      rq_wait_ft_sensor_steady(2000)
      zero_ftsensor()
      sleep(0.1)
      # end: URCap Program Node
      # begin: URCap Program Node
      #   Source: Robotiq_Copilot, 1.22.1.14215, Robotiq Inc.
      #   Type: Finishing Tool Control
      $ 59 "Start tool"
      set_standard_digital_out(3, True)
      # end: URCap Program Node
      $ 60 "If dried2≟ False "
      if (dried2 ==   False  ):
        $ 61 "Force"
        sleep(0.02)
        zero_ftsensor()
        force_mode(p[0.0,0.0,0.0,0.0,0.0,0.0], [0, 0, 1, 0, 0, 0], [0.0, 0.0, 6.0, 0.0, 0.0, 0.0], 2, [0.1, 0.1, 0.15, 0.3490658503988659, 0.3490658503988659, 0.3490658503988659])
        $ 62 "Conveyor_Move_mm(width-12)" "noBreak"
        Conveyor_Move_mm(width-12)
        $ 63 "Wait SERVER_STATE==1" "noBreak"
        while (not(modbus_get_signal_status("SERVER_STATE")==1)):
          sync()
        end
        $ 64 "moveHeight" "noBreak"
        $ 65 "currentPosition≔get_actual_tcp_pose()" "noBreak"
        global currentPosition=get_actual_tcp_pose()
        $ 66 "newPosition≔pose_add(currentPosition, p[-height/1000,0,0,0,0,0])" "noBreak"
        global newPosition=pose_add(currentPosition, p[-height/1000,0,0,0,0,0])
        $ 67 "newPosition" "noBreak"
        movel(newPosition, a=0.5, v=0.05)
        $ 68 "Conveyor_Move_mm(-width+12)" "noBreak"
        Conveyor_Move_mm(-width+12)
        $ 69 "Wait SERVER_STATE==1" "noBreak"
        while (not(modbus_get_signal_status("SERVER_STATE")==1)):
          sync()
        end
        $ 70 "moveHeight" "noBreak"
        $ 71 "currentPosition≔get_actual_tcp_pose()" "noBreak"
        global currentPosition=get_actual_tcp_pose()
        $ 72 "newPosition≔pose_add(currentPosition, p[height/1000,0,0,0,0,0])" "noBreak"
        global newPosition=pose_add(currentPosition, p[height/1000,0,0,0,0,0])
        $ 73 "newPosition" "noBreak"
        movel(newPosition, a=0.5, v=0.05)
        # begin: URCap Program Node
        #   Source: Robotiq_Copilot, 1.22.1.14215, Robotiq Inc.
        #   Type: Finishing Tool Control
        $ 74 "Stop tool" "noBreak"
        set_standard_digital_out(3, False)
        # end: URCap Program Node
        end_force_mode()
        stopl(5.0)
      else:
        $ 75 "Else" "noBreak"
        $ 76 "Force"
        sleep(0.02)
        zero_ftsensor()
        force_mode(p[0.0,0.0,0.0,0.0,0.0,0.0], [0, 0, 1, 0, 0, 0], [0.0, 0.0, 6.0, 0.0, 0.0, 0.0], 2, [0.1, 0.1, 0.15, 0.3490658503988659, 0.3490658503988659, 0.3490658503988659])
        $ 77 "Conveyor_Move_mm(width-12)" "noBreak"
        Conveyor_Move_mm(width-12)
        $ 78 "Wait SERVER_STATE==1" "noBreak"
        while (not(modbus_get_signal_status("SERVER_STATE")==1)):
          sync()
        end
        $ 79 "moveHeight" "noBreak"
        $ 80 "currentPosition≔get_actual_tcp_pose()" "noBreak"
        global currentPosition=get_actual_tcp_pose()
        $ 81 "newPosition≔pose_add(currentPosition, p[-height/1000,0,0,0,0,0])" "noBreak"
        global newPosition=pose_add(currentPosition, p[-height/1000,0,0,0,0,0])
        $ 82 "newPosition" "noBreak"
        movel(newPosition, a=0.5, v=0.05)
        $ 83 "Conveyor_Move_mm(-width+12)" "noBreak"
        Conveyor_Move_mm(-width+12)
        $ 84 "Wait SERVER_STATE==1" "noBreak"
        while (not(modbus_get_signal_status("SERVER_STATE")==1)):
          sync()
        end
        $ 85 "moveHeight" "noBreak"
        $ 86 "currentPosition≔get_actual_tcp_pose()" "noBreak"
        global currentPosition=get_actual_tcp_pose()
        $ 87 "newPosition≔pose_add(currentPosition, p[height/1000,0,0,0,0,0])" "noBreak"
        global newPosition=pose_add(currentPosition, p[height/1000,0,0,0,0,0])
        $ 88 "newPosition" "noBreak"
        movel(newPosition, a=0.5, v=0.05)
        # begin: URCap Program Node
        #   Source: Robotiq_Copilot, 1.22.1.14215, Robotiq Inc.
        #   Type: Finishing Tool Control
        $ 89 "Stop tool" "noBreak"
        set_standard_digital_out(3, False)
        # end: URCap Program Node
        end_force_mode()
        stopl(5.0)
      end
      $ 90 "MoveJ"
      $ 91 "Sand_Base" "breakAfter"
      movej(get_inverse_kin(Sand_Base_p, qnear=Sand_Base_q), a=1.3962634015954636, v=1.0471975511965976)
      $ 92 "45 Sand"
      $ 93 "If JOB == 3"
      if (modbus_get_signal_status("JOB") == 3):
        $ 94 "Conveyor_Move_mm((width-12)/3)"
        Conveyor_Move_mm((width-12)/3)
        $ 95 "Wait SERVER_STATE==1"
        while (not(modbus_get_signal_status("SERVER_STATE")==1)):
          sync()
        end
        $ 96 "MoveL"
        $ 97 "Direction: Base Z+"
        global move_thread_flag_97=0
        thread move_thread_97():
          enter_critical
          move_thread_flag_97 = 1
          local towardsPos=calculate_point_to_move_towards(p[0.0,0.0,0.0,0.0,0.0,0.0], [0.0,0.0,1.0], 1000.0)
          movel(towardsPos, a=0.5, v=0.05)
          move_thread_flag_97 = 2
          exit_critical
        end
        move_thread_flag_97 = 0
        move_thread_han_97 = run move_thread_97()
        while (True):
          local targetTcpDirection=get_target_tcp_speed()
          local stepsToRetract=tool_contact(direction=targetTcpDirection)
          if (stepsToRetract > 0):
            kill move_thread_han_97
            stopl(3.0)
            local backTrackMovement=get_actual_joint_positions_history(stepsToRetract)
            local contactPose=get_forward_kin(backTrackMovement)
            local posDir=[targetTcpDirection[0],targetTcpDirection[1],targetTcpDirection[2]]
            local retractTo=contactPose
            if (norm(posDir) > 1e-6):
              local normalizedPosDir=normalize(posDir)
              local additionalRetraction=p[normalizedPosDir[0] * 0.0, normalizedPosDir[1] * 0.0, normalizedPosDir[2] * 0.0, 0, 0, 0]
              retractTo = pose_sub(contactPose, additionalRetraction)
            end
            movel(retractTo, a=3.0, v=0.1)
            $ 98 "Until (tool_contact_detection)"
            break
          end
          sync()
        end
        # begin: URCap Program Node
        #   Source: Robotiq_Copilot, 1.22.1.14215, Robotiq Inc.
        #   Type: Finishing Tool Control
        $ 99 "Start tool"
        set_standard_digital_out(3, True)
        # end: URCap Program Node
        $ 100 "Force"
        sleep(0.02)
        zero_ftsensor()
        force_mode(p[0.0,0.0,0.0,0.0,0.0,0.0], [0, 0, 1, 0, 0, 0], [0.0, 0.0, 7.0, 0.0, 0.0, 0.0], 2, [0.1, 0.1, 0.15, 0.3490658503988659, 0.3490658503988659, 0.3490658503988659])
        $ 101 "moveHeight" "noBreak"
        $ 102 "currentPosition≔get_actual_tcp_pose()" "noBreak"
        global currentPosition=get_actual_tcp_pose()
        $ 103 "newPosition≔pose_add(currentPosition, p[-height/1000,0,0,0,0,0])" "noBreak"
        global newPosition=pose_add(currentPosition, p[-height/1000,0,0,0,0,0])
        $ 104 "newPosition" "noBreak"
        set_tcp(p[0.0010032816279412216,0.1255407840271643,0.10415400799666161,-0.7853981633974483,0.0,0.0])
        movel(newPosition, a=0.5, v=0.05)
        # begin: URCap Program Node
        #   Source: Robotiq_Copilot, 1.22.1.14215, Robotiq Inc.
        #   Type: Finishing Tool Control
        $ 105 "Stop tool" "noBreak"
        set_standard_digital_out(3, False)
        # end: URCap Program Node
        end_force_mode()
        stopl(5.0)
        $ 106 "Direction: Base Z-"
        global move_thread_flag_106=0
        thread move_thread_106():
          enter_critical
          move_thread_flag_106 = 1
          local towardsPos=calculate_point_to_move_towards(p[0.0,0.0,0.0,0.0,0.0,0.0], [0.0,0.0,-1.0], 0.02)
          movel(towardsPos, a=0.5, v=0.05)
          move_thread_flag_106 = 2
          exit_critical
        end
        move_thread_flag_106 = 0
        move_thread_han_106 = run move_thread_106()
        while (True):
          sleep(1.0E-10)
          if (move_thread_flag_106 > 1):
            join move_thread_han_106
            $ 107 "Until (distance)"
            break
          end
          sync()
        end
        $ 108 "Conveyor_Move_mm((width-12)/3)"
        Conveyor_Move_mm((width-12)/3)
        $ 109 "Wait SERVER_STATE==1"
        while (not(modbus_get_signal_status("SERVER_STATE")==1)):
          sync()
        end
        $ 110 "Direction: Base Z+"
        global move_thread_flag_110=0
        thread move_thread_110():
          enter_critical
          move_thread_flag_110 = 1
          local towardsPos=calculate_point_to_move_towards(p[0.0,0.0,0.0,0.0,0.0,0.0], [0.0,0.0,1.0], 1000.0)
          movel(towardsPos, a=0.5, v=0.05)
          move_thread_flag_110 = 2
          exit_critical
        end
        move_thread_flag_110 = 0
        move_thread_han_110 = run move_thread_110()
        while (True):
          local targetTcpDirection=get_target_tcp_speed()
          local stepsToRetract=tool_contact(direction=targetTcpDirection)
          if (stepsToRetract > 0):
            kill move_thread_han_110
            stopl(3.0)
            local backTrackMovement=get_actual_joint_positions_history(stepsToRetract)
            local contactPose=get_forward_kin(backTrackMovement)
            local posDir=[targetTcpDirection[0],targetTcpDirection[1],targetTcpDirection[2]]
            local retractTo=contactPose
            if (norm(posDir) > 1e-6):
              local normalizedPosDir=normalize(posDir)
              local additionalRetraction=p[normalizedPosDir[0] * 0.0, normalizedPosDir[1] * 0.0, normalizedPosDir[2] * 0.0, 0, 0, 0]
              retractTo = pose_sub(contactPose, additionalRetraction)
            end
            movel(retractTo, a=3.0, v=0.1)
            $ 111 "Until (tool_contact_detection)"
            break
          end
          sync()
        end
        $ 112 "Force"
        sleep(0.02)
        zero_ftsensor()
        force_mode(p[0.0,0.0,0.0,0.0,0.0,0.0], [0, 0, 1, 0, 0, 0], [0.0, 0.0, 7.0, 0.0, 0.0, 0.0], 2, [0.1, 0.1, 0.15, 0.3490658503988659, 0.3490658503988659, 0.3490658503988659])
        # begin: URCap Program Node
        #   Source: Robotiq_Copilot, 1.22.1.14215, Robotiq Inc.
        #   Type: Finishing Tool Control
        $ 113 "Start tool" "noBreak"
        set_standard_digital_out(3, True)
        # end: URCap Program Node
        $ 114 "moveHeight" "noBreak"
        $ 115 "currentPosition≔get_actual_tcp_pose()" "noBreak"
        global currentPosition=get_actual_tcp_pose()
        $ 116 "newPosition≔pose_add(currentPosition, p[height/1000,0,0,0,0,0])" "noBreak"
        global newPosition=pose_add(currentPosition, p[height/1000,0,0,0,0,0])
        $ 117 "newPosition" "noBreak"
        set_tcp(p[0.0010032816279412216,0.1255407840271643,0.10415400799666161,-0.7853981633974483,0.0,0.0])
        movel(newPosition, a=0.5, v=0.05)
        # begin: URCap Program Node
        #   Source: Robotiq_Copilot, 1.22.1.14215, Robotiq Inc.
        #   Type: Finishing Tool Control
        $ 118 "Stop tool" "noBreak"
        set_standard_digital_out(3, False)
        # end: URCap Program Node
        end_force_mode()
        stopl(5.0)
        $ 119 "Direction: Base Z-"
        global move_thread_flag_119=0
        thread move_thread_119():
          enter_critical
          move_thread_flag_119 = 1
          local towardsPos=calculate_point_to_move_towards(p[0.0,0.0,0.0,0.0,0.0,0.0], [0.0,0.0,-1.0], 0.02)
          movel(towardsPos, a=0.5, v=0.05)
          move_thread_flag_119 = 2
          exit_critical
        end
        move_thread_flag_119 = 0
        move_thread_han_119 = run move_thread_119()
        while (True):
          sleep(1.0E-10)
          if (move_thread_flag_119 > 1):
            join move_thread_han_119
            $ 120 "Until (distance)"
            break
          end
          sync()
        end
        $ 121 "Conveyor_Move_mm(-(width-12)*2/3)"
        Conveyor_Move_mm(-(width-12)*2/3)
        $ 122 "Wait SERVER_STATE==1"
        while (not(modbus_get_signal_status("SERVER_STATE")==1)):
          sync()
        end
      end
      $ 123 "SC 3 and 4 Sand"
      $ 124 "If JOB == 5 or JOB == 6"
      if (modbus_get_signal_status("JOB") == 5 or modbus_get_signal_status("JOB") == 6):
        $ 125 "Conveyor_Move_mm((width-12)/2)"
        Conveyor_Move_mm((width-12)/2)
        $ 126 "Wait SERVER_STATE==1"
        while (not(modbus_get_signal_status("SERVER_STATE")==1)):
          sync()
        end
        $ 127 "MoveL"
        $ 128 "Direction: Base X-"
        global move_thread_flag_128=0
        thread move_thread_128():
          enter_critical
          move_thread_flag_128 = 1
          local towardsPos=calculate_point_to_move_towards(p[0.0,0.0,0.0,0.0,0.0,0.0], [-1.0,0.0,0.0], 0.085)
          movel(towardsPos, a=0.5, v=0.05)
          move_thread_flag_128 = 2
          exit_critical
        end
        move_thread_flag_128 = 0
        move_thread_han_128 = run move_thread_128()
        while (True):
          sleep(1.0E-10)
          if (move_thread_flag_128 > 1):
            join move_thread_han_128
            $ 129 "Until (distance)"
            break
          end
          sync()
        end
        $ 130 "Direction: Base Z+"
        global move_thread_flag_130=0
        thread move_thread_130():
          enter_critical
          move_thread_flag_130 = 1
          local towardsPos=calculate_point_to_move_towards(p[0.0,0.0,0.0,0.0,0.0,0.0], [0.0,0.0,1.0], 1000.0)
          movel(towardsPos, a=0.5, v=0.05)
          move_thread_flag_130 = 2
          exit_critical
        end
        move_thread_flag_130 = 0
        move_thread_han_130 = run move_thread_130()
        while (True):
          local targetTcpDirection=get_target_tcp_speed()
          local stepsToRetract=tool_contact(direction=targetTcpDirection)
          if (stepsToRetract > 0):
            kill move_thread_han_130
            stopl(3.0)
            local backTrackMovement=get_actual_joint_positions_history(stepsToRetract)
            local contactPose=get_forward_kin(backTrackMovement)
            local posDir=[targetTcpDirection[0],targetTcpDirection[1],targetTcpDirection[2]]
            local retractTo=contactPose
            if (norm(posDir) > 1e-6):
              local normalizedPosDir=normalize(posDir)
              local additionalRetraction=p[normalizedPosDir[0] * 0.0, normalizedPosDir[1] * 0.0, normalizedPosDir[2] * 0.0, 0, 0, 0]
              retractTo = pose_sub(contactPose, additionalRetraction)
            end
            movel(retractTo, a=3.0, v=0.1)
            $ 131 "Until (tool_contact_detection)"
            break
          end
          sync()
        end
        # begin: URCap Program Node
        #   Source: Robotiq_Copilot, 1.22.1.14215, Robotiq Inc.
        #   Type: Finishing Tool Control
        $ 132 "Start tool"
        set_standard_digital_out(3, True)
        # end: URCap Program Node
        $ 133 "Force"
        sleep(0.02)
        zero_ftsensor()
        force_mode(p[0.0,0.0,0.0,0.0,0.0,0.0], [0, 0, 1, 0, 0, 0], [0.0, 0.0, 10.0, 0.0, 0.0, 0.0], 2, [0.1, 0.1, 0.15, 0.3490658503988659, 0.3490658503988659, 0.3490658503988659])
        $ 134 "Direction: Base X-" "noBreak"
        global move_thread_flag_134=0
        thread move_thread_134():
          enter_critical
          move_thread_flag_134 = 1
          local towardsPos=calculate_point_to_move_towards(p[0.0,0.0,0.0,0.0,0.0,0.0], [-1.0,0.0,0.0], 0.08)
          movel(towardsPos, a=0.5, v=0.05)
          move_thread_flag_134 = 2
          exit_critical
        end
        move_thread_flag_134 = 0
        move_thread_han_134 = run move_thread_134()
        while (True):
          sleep(1.0E-10)
          if (move_thread_flag_134 > 1):
            join move_thread_han_134
            $ 135 "Until (distance)" "noBreak"
            break
          end
          sync()
        end
        # begin: URCap Program Node
        #   Source: Robotiq_Copilot, 1.22.1.14215, Robotiq Inc.
        #   Type: Finishing Tool Control
        $ 136 "Stop tool" "noBreak"
        set_standard_digital_out(3, False)
        # end: URCap Program Node
        end_force_mode()
        stopl(5.0)
        $ 137 "Direction: Base Z-"
        global move_thread_flag_137=0
        thread move_thread_137():
          enter_critical
          move_thread_flag_137 = 1
          local towardsPos=calculate_point_to_move_towards(p[0.0,0.0,0.0,0.0,0.0,0.0], [0.0,0.0,-1.0], 0.05)
          movel(towardsPos, a=0.5, v=0.05)
          move_thread_flag_137 = 2
          exit_critical
        end
        move_thread_flag_137 = 0
        move_thread_han_137 = run move_thread_137()
        while (True):
          sleep(1.0E-10)
          if (move_thread_flag_137 > 1):
            join move_thread_han_137
            $ 138 "Until (distance)"
            break
          end
          sync()
        end
        $ 139 "Conveyor_Move_mm(-(width-12)/2)"
        Conveyor_Move_mm(-(width-12)/2)
        $ 140 "Wait SERVER_STATE==1"
        while (not(modbus_get_signal_status("SERVER_STATE")==1)):
          sync()
        end
      end
      $ 141 "Spray Vertical"
      $ 142 "MoveJ"
      $ 143 "Spray_Base" "breakAfter"
      set_tcp(p[0.06314273891748035,-0.10788249600106846,0.08439511317031662,0.6139431255689367,0.6139431255689367,-1.4821898202742554])
      movej(get_inverse_kin(Spray_Base_p, qnear=Spray_Base_q), a=1.3962634015954636, v=1.0471975511965976)
      $ 144 "If JOB == 2"
      if (modbus_get_signal_status("JOB") == 2):
        $ 145 "MoveL"
        $ 146 "Direction: Base Z+"
        global move_thread_flag_146=0
        thread move_thread_146():
          enter_critical
          move_thread_flag_146 = 1
          local towardsPos=calculate_point_to_move_towards(p[0.0,0.0,0.0,0.0,0.0,0.0], [0.0,0.0,1.0], 0.1)
          movel(towardsPos, a=1.2, v=0.25)
          move_thread_flag_146 = 2
          exit_critical
        end
        move_thread_flag_146 = 0
        move_thread_han_146 = run move_thread_146()
        while (True):
          sleep(1.0E-10)
          if (move_thread_flag_146 > 1):
            join move_thread_han_146
            $ 147 "Until (distance)"
            break
          end
          sync()
        end
      end
      $ 148 "If JOB == 7"
      if (modbus_get_signal_status("JOB") == 7):
        $ 149 "MoveL"
        $ 150 "Direction: Base Z+"
        global move_thread_flag_150=0
        thread move_thread_150():
          enter_critical
          move_thread_flag_150 = 1
          local towardsPos=calculate_point_to_move_towards(p[0.0,0.0,0.0,0.0,0.0,0.0], [0.0,0.0,1.0], 0.2)
          movel(towardsPos, a=1.2, v=0.25)
          move_thread_flag_150 = 2
          exit_critical
        end
        move_thread_flag_150 = 0
        move_thread_han_150 = run move_thread_150()
        while (True):
          sleep(1.0E-10)
          if (move_thread_flag_150 > 1):
            join move_thread_han_150
            $ 151 "Until (distance)"
            break
          end
          sync()
        end
      end
      $ 152 "Set SprayerOn=On"
      set_standard_digital_out(5, True)
      $ 153 "MoveL"
      $ 154 "Conveyor_Move_mm(width-12)"
      Conveyor_Move_mm(width-12)
      $ 155 "Wait SERVER_STATE==1"
      while (not(modbus_get_signal_status("SERVER_STATE")==1)):
        sync()
      end
      $ 156 "moveHeight"
      $ 157 "currentPosition≔get_actual_tcp_pose()"
      global currentPosition=get_actual_tcp_pose()
      $ 158 "newPosition≔pose_add(currentPosition, p[-height/1000,0,0,0,0,0])"
      global newPosition=pose_add(currentPosition, p[-height/1000,0,0,0,0,0])
      $ 159 "newPosition" "breakAfter"
      movel(newPosition, a=0.5, v=0.05)
      $ 160 "Conveyor_Move_mm(-width+12)"
      Conveyor_Move_mm(-width+12)
      $ 161 "Wait SERVER_STATE==1"
      while (not(modbus_get_signal_status("SERVER_STATE")==1)):
        sync()
      end
      $ 162 "moveHeight"
      $ 163 "currentPosition≔get_actual_tcp_pose()"
      global currentPosition=get_actual_tcp_pose()
      $ 164 "newPosition≔pose_add(currentPosition, p[height/1000,0,0,0,0,0])"
      global newPosition=pose_add(currentPosition, p[height/1000,0,0,0,0,0])
      $ 165 "newPosition" "breakAfter"
      movel(newPosition, a=0.5, v=0.05)
      $ 166 "Set SprayerOn=Off"
      set_standard_digital_out(5, False)
      $ 167 "MoveJ"
      $ 168 "Spray_Base" "breakAfter"
      movej(get_inverse_kin(Spray_Base_p, qnear=Spray_Base_q), a=1.3962634015954636, v=1.0471975511965976)
      $ 169 "45 Spray"
      $ 170 "If JOB == 3"
      if (modbus_get_signal_status("JOB") == 3):
        $ 171 "MoveJ"
        $ 172 "Spray_Base" "breakAfter"
        set_tcp(p[0.06314273891748035,-0.10788249600106846,0.08439511317031662,0.6139431255689367,0.6139431255689367,-1.4821898202742554])
        movej(get_inverse_kin(Spray_Base_p, qnear=Spray_Base_q), a=1.3962634015954636, v=1.0471975511965976)
        $ 173 "MoveL"
        $ 174 "Conveyor_Move_mm(width/3)"
        Conveyor_Move_mm(width/3)
        $ 175 "Wait SERVER_STATE==1"
        while (not(modbus_get_signal_status("SERVER_STATE")==1)):
          sync()
        end
        $ 176 "Set SprayerOn=On"
        set_standard_digital_out(5, True)
        $ 177 "moveHeight"
        $ 178 "currentPosition≔get_actual_tcp_pose()"
        global currentPosition=get_actual_tcp_pose()
        $ 179 "newPosition≔pose_add(currentPosition, p[-height/1000,0,0,0,0,0])"
        global newPosition=pose_add(currentPosition, p[-height/1000,0,0,0,0,0])
        $ 180 "newPosition" "breakAfter"
        movel(newPosition, a=0.5, v=0.05)
        $ 181 "Set SprayerOn=Off"
        set_standard_digital_out(5, False)
        $ 182 "Conveyor_Move_mm(width/3)"
        Conveyor_Move_mm(width/3)
        $ 183 "Wait SERVER_STATE==1"
        while (not(modbus_get_signal_status("SERVER_STATE")==1)):
          sync()
        end
        $ 184 "Set SprayerOn=On"
        set_standard_digital_out(5, True)
        $ 185 "moveHeight"
        $ 186 "currentPosition≔get_actual_tcp_pose()"
        global currentPosition=get_actual_tcp_pose()
        $ 187 "newPosition≔pose_add(currentPosition, p[height/1000,0,0,0,0,0])"
        global newPosition=pose_add(currentPosition, p[height/1000,0,0,0,0,0])
        $ 188 "newPosition" "breakAfter"
        movel(newPosition, a=0.5, v=0.05)
        $ 189 "Set SprayerOn=Off"
        set_standard_digital_out(5, False)
        $ 190 "MoveJ"
        $ 191 "Spray_Base" "breakAfter"
        movej(get_inverse_kin(Spray_Base_p, qnear=Spray_Base_q), a=1.3962634015954636, v=1.0471975511965976)
      end
      $ 192 "SC 3 and 4 Spray"
      $ 193 "If JOB == 5 or JOB == 6"
      if (modbus_get_signal_status("JOB") == 5 or modbus_get_signal_status("JOB") == 6):
        $ 194 "MoveJ"
        $ 195 "Spray_Base" "breakAfter"
        set_tcp(p[0.06314273891748035,-0.10788249600106846,0.08439511317031662,0.6139431255689367,0.6139431255689367,-1.4821898202742554])
        movej(get_inverse_kin(Spray_Base_p, qnear=Spray_Base_q), a=1.3962634015954636, v=1.0471975511965976)
        $ 196 "Conveyor_Move_mm((width-12)/2)"
        Conveyor_Move_mm((width-12)/2)
        $ 197 "Wait SERVER_STATE==1"
        while (not(modbus_get_signal_status("SERVER_STATE")==1)):
          sync()
        end
        $ 198 "MoveL"
        $ 199 "Direction: Base X-"
        global move_thread_flag_199=0
        thread move_thread_199():
          enter_critical
          move_thread_flag_199 = 1
          local towardsPos=calculate_point_to_move_towards(p[0.0,0.0,0.0,0.0,0.0,0.0], [-1.0,0.0,0.0], 0.012)
          movel(towardsPos, a=0.5, v=0.05)
          move_thread_flag_199 = 2
          exit_critical
        end
        move_thread_flag_199 = 0
        move_thread_han_199 = run move_thread_199()
        while (True):
          sleep(1.0E-10)
          if (move_thread_flag_199 > 1):
            join move_thread_han_199
            $ 200 "Until (distance)"
            break
          end
          sync()
        end
        $ 201 "Set SprayerOn=On"
        set_standard_digital_out(5, True)
        $ 202 "Direction: Base X-"
        global move_thread_flag_202=0
        thread move_thread_202():
          enter_critical
          move_thread_flag_202 = 1
          local towardsPos=calculate_point_to_move_towards(p[0.0,0.0,0.0,0.0,0.0,0.0], [-1.0,0.0,0.0], 0.21)
          movel(towardsPos, a=0.5, v=0.05)
          move_thread_flag_202 = 2
          exit_critical
        end
        move_thread_flag_202 = 0
        move_thread_han_202 = run move_thread_202()
        while (True):
          sleep(1.0E-10)
          if (move_thread_flag_202 > 1):
            join move_thread_han_202
            $ 203 "Until (distance)"
            break
          end
          sync()
        end
        $ 204 "Set SprayerOn=Off"
        set_standard_digital_out(5, False)
        $ 205 "Conveyor_Move_mm(-(width-12)/2)"
        Conveyor_Move_mm(-(width-12)/2)
        $ 206 "Wait SERVER_STATE==1"
        while (not(modbus_get_signal_status("SERVER_STATE")==1)):
          sync()
        end
      end
      $ 207 "Cube"
      $ 208 "If JOB==1"
      if (modbus_get_signal_status("JOB")==1):
        $ 209 "Spray Horizontal"
        $ 210 "MoveJ"
        $ 211 "Waypoint_1" "breakAfter"
        set_tcp(p[0.06314273891748035,-0.10788249600106846,0.08439511317031662,0.6139431255689367,0.6139431255689367,-1.4821898202742554])
        movej(get_inverse_kin(Waypoint_1_p, qnear=Waypoint_1_q), a=1.3962634015954636, v=1.0471975511965976)
        $ 212 "Set SprayerOn=On"
        set_standard_digital_out(5, True)
        $ 213 "Conveyor_Move_mm(width-12)"
        Conveyor_Move_mm(width-12)
        $ 214 "Wait SERVER_STATE==1"
        while (not(modbus_get_signal_status("SERVER_STATE")==1)):
          sync()
        end
        $ 215 "Set SprayerOn=Off"
        set_standard_digital_out(5, False)
        $ 216 "Waypoint_2" "breakAfter"
        set_tcp(p[0.06314273891748035,-0.10788249600106846,0.08439511317031662,0.6139431255689367,0.6139431255689367,-1.4821898202742554])
        movej(get_inverse_kin(Waypoint_2_p, qnear=Waypoint_2_q), a=1.3962634015954636, v=1.0471975511965976)
        $ 217 "MoveL"
        $ 218 "Set SprayerOn=On"
        set_standard_digital_out(5, True)
        $ 219 "moveHeight"
        $ 220 "currentPosition≔get_actual_tcp_pose()"
        global currentPosition=get_actual_tcp_pose()
        $ 221 "newPosition≔pose_add(currentPosition, p[-height/1000,0,0,0,0,0])"
        global newPosition=pose_add(currentPosition, p[-height/1000,0,0,0,0,0])
        $ 222 "newPosition" "breakAfter"
        movel(newPosition, a=0.5, v=0.05)
        $ 223 "Set SprayerOn=Off"
        set_standard_digital_out(5, False)
        $ 224 "Conveyor_Move_mm(-width+12)"
        Conveyor_Move_mm(-width+12)
        $ 225 "Waypoint_3" "breakAfter"
        set_tcp(p[0.06314273891748035,-0.10788249600106846,0.08439511317031662,0.6139431255689367,0.6139431255689367,-1.4821898202742554])
        movej(get_inverse_kin(Waypoint_3_p, qnear=Waypoint_3_q), a=1.3962634015954636, v=1.0471975511965976)
        $ 226 "Wait SERVER_STATE==1"
        while (not(modbus_get_signal_status("SERVER_STATE")==1)):
          sync()
        end
        $ 227 "MoveL"
        $ 228 "Set SprayerOn=On"
        set_standard_digital_out(5, True)
        $ 229 "moveHeight"
        $ 230 "currentPosition≔get_actual_tcp_pose()"
        global currentPosition=get_actual_tcp_pose()
        $ 231 "newPosition≔pose_add(currentPosition, p[height/1000,0,0,0,0,0])"
        global newPosition=pose_add(currentPosition, p[height/1000,0,0,0,0,0])
        $ 232 "newPosition" "breakAfter"
        movel(newPosition, a=0.5, v=0.05)
        $ 233 "Set SprayerOn=Off"
        set_standard_digital_out(5, False)
      end
      $ 234 "MoveJ"
      $ 235 "Sand_Base" "breakAfter"
      set_tcp(p[0.0010032816279412216,0.1255407840271643,0.10415400799666161,-0.7853981633974483,0.0,0.0])
      movej(get_inverse_kin(Sand_Base_p, qnear=Sand_Base_q), a=1.3962634015954636, v=1.0471975511965976)
      $ 236 "Clean Spray"
      $ 237 "MoveJ"
      $ 238 "Sand_Base" "breakAfter"
      set_tcp(p[0.0010032816279412216,0.1255407840271643,0.10415400799666161,-0.7853981633974483,0.0,0.0])
      movej(get_inverse_kin(Sand_Base_p, qnear=Sand_Base_q), a=1.3962634015954636, v=1.0471975511965976)
      $ 239 "Clean_Brush" "breakAfter"
      set_tcp(p[0.0010032816279412216,0.1255407840271643,0.10415400799666161,-0.7853981633974483,0.0,0.0])
      movej(get_inverse_kin(Clean_Brush_p, qnear=Clean_Brush_q), a=1.3962634015954636, v=1.0471975511965976)
      $ 240 "MoveL"
      $ 241 "Direction: Base Z+"
      global move_thread_flag_241=0
      thread move_thread_241():
        enter_critical
        move_thread_flag_241 = 1
        local towardsPos=calculate_point_to_move_towards(p[0.0,0.0,0.0,0.0,0.0,0.0], [0.0,0.0,1.0], 1000.0)
        movel(towardsPos, a=0.5, v=0.05)
        move_thread_flag_241 = 2
        exit_critical
      end
      move_thread_flag_241 = 0
      move_thread_han_241 = run move_thread_241()
      while (True):
        local targetTcpDirection=get_target_tcp_speed()
        local stepsToRetract=tool_contact(direction=targetTcpDirection)
        if (stepsToRetract > 0):
          kill move_thread_han_241
          stopl(0.5)
          local backTrackMovement=get_actual_joint_positions_history(stepsToRetract)
          local contactPose=get_forward_kin(backTrackMovement)
          local posDir=[targetTcpDirection[0],targetTcpDirection[1],targetTcpDirection[2]]
          local retractTo=contactPose
          if (norm(posDir) > 1e-6):
            local normalizedPosDir=normalize(posDir)
            local additionalRetraction=p[normalizedPosDir[0] * 0.003, normalizedPosDir[1] * 0.003, normalizedPosDir[2] * 0.003, 0, 0, 0]
            retractTo = pose_sub(contactPose, additionalRetraction)
          end
          movel(retractTo, a=0.5, v=0.1)
          $ 242 "Until (tool_contact_detection)"
          break
        end
        sync()
      end
      $ 243 "Wait: 1.0"
      sleep(1.0)
      $ 244 "Set BRUSH_ON_LOCAL= True "
      modbus_set_output_signal("BRUSH_ON_LOCAL",   True  )
      $ 245 "timer_brush: Start"
      timer_brush_is_counting = True
      $ 246 "If dried2≟ False "
      if (dried2 ==   False  ):
        $ 247 "Dry"
        $ 248 "timer_dry: Start"
        timer_dry_is_counting = True
        $ 249 "Conveyor_Move_mm(width+500)"
        Conveyor_Move_mm(width+500)
        $ 250 "Wait SERVER_STATE==1"
        while (not(modbus_get_signal_status("SERVER_STATE")==1)):
          sync()
        end
        $ 251 "Loop timer_dry<165"
        while (timer_dry<165):
          $ 252 "Conveyor_Move_mm(-(width/2))"
          Conveyor_Move_mm(-(width/2))
          $ 253 "Wait SERVER_STATE==1"
          while (not(modbus_get_signal_status("SERVER_STATE")==1)):
            sync()
          end
          $ 254 "Conveyor_Move_mm(width/2)"
          Conveyor_Move_mm(width/2)
          $ 255 "Wait SERVER_STATE==1"
          while (not(modbus_get_signal_status("SERVER_STATE")==1)):
            sync()
          end
        end
        $ 256 "Move_Continuous('reverse')"
        Move_Continuous("reverse")
        $ 257 "Wait WORK_AT_ZERO=HI"
        while (modbus_get_signal_status("WORK_AT_ZERO") == False):
          sync()
        end
        $ 258 "Wait WORK_AT_ZERO=LO"
        while (modbus_get_signal_status("WORK_AT_ZERO") == True):
          sync()
        end
        $ 259 "Move_Continuous('forward')"
        Move_Continuous("forward")
        $ 260 "Wait WORK_AT_ZERO=HI"
        while (modbus_get_signal_status("WORK_AT_ZERO") == False):
          sync()
        end
        $ 261 "dried2≔ True "
        global dried2=  True
        $ 262 "timer_dry: Stop"
        timer_dry_is_counting = False
        $ 263 "timer_dry: Reset"
        timer_dry = 0
        $ 264 "Move_Idle()"
        Move_Idle()
      else:
        $ 265 "Else" "noBreak"
        $ 266 "Unload Workpiece"
        $ 267 "Move_Continuous('forward')"
        Move_Continuous("forward")
        $ 268 "Wait OFFLOAD=HI"
        while (modbus_get_signal_status("OFFLOAD") == False):
          sync()
        end
        $ 269 "Wait OFFLOAD=LO"
        while (modbus_get_signal_status("OFFLOAD") == True):
          sync()
        end
        $ 270 "loaded≔0"
        global loaded=0
        $ 271 "dried2≔ False "
        global dried2=  False
        $ 272 "Wait: 1.0"
        sleep(1.0)
        $ 273 "Move_Idle()"
        Move_Idle()
      end
    end
    $ 280 "sync()"
    sync()
  end
end
